Staubli VAL3: onEnterEvent.pgx

program onEnterEvent()
begin
  //
end
